PROGRAM pouPROFINETdiag
VAR
	iVal: WORD;
	tVal: WORD;
	tmask: WORD;
	state: UINT;
	i: UINT;
	decode:fb_decodeProfiNet;
	
	retvall: UDINT;
	idbGetConfSlaves: FB_EcGetConfSlaves;
	test: BOOL;
	testams: BOOL;
	a: UINT;
	tDiagScreenSize: UINT;
	tDiagScreenWidth: UINT;
	tDiagScreenPointer: UINT;
	testvalprofinet: PROFINETstate;
	
	detectFallingFault:F_TRIG;
END_VAR
VAR // added by the converter: edge detectors and wires of the graphical bodies
    _rt1, _rt2, _rt3, _rt4, _rt5 : R_TRIG;
END_VAR

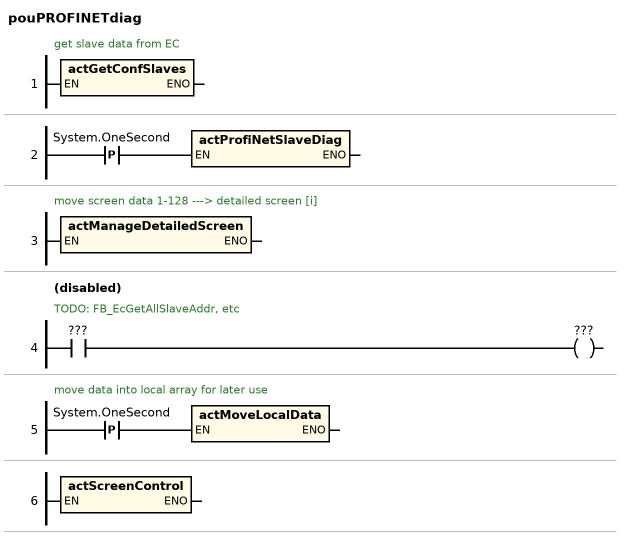
// NETWORK 1
// get slave data from EC
actGetConfSlaves();

// NETWORK 2
_rt1(CLK := System.OneSecond);
IF _rt1.Q THEN actProfiNetSlaveDiag(); END_IF

// NETWORK 3
// move screen data 1-128 ---> detailed screen [i]
actManageDetailedScreen();

// NETWORK 4 (disabled)
// TODO: FB_EcGetAllSlaveAddr, etc
// ??? := ???;

// NETWORK 5
// move data into local array for later use
_rt2(CLK := System.OneSecond);
IF _rt2.Q THEN actMoveLocalData(); END_IF

// NETWORK 6
actScreenControl();

ACTION actGetConfSlaves:
// NETWORK 1
// use System.OneSecond to slow down reading

// NETWORK 2
// get additional profinet info via ADS
END_ACTION

ACTION actManageDetailedScreen:
//get max value of diag number
ProfiNetDiag.detailDiagNum := MAX(ProfiNetDiag.detailDiagNum, 1);

IF System.PulseOneSecond THEN
	retvall := MEMCPY( destAddr	:=ADR(ProfiNetDiag.detailDiag),
						srcAddr :=ADR(ProfiNetDiag.diagScreen[ProfiNetDiag.detailDiagNum]),
						n		:=SIZEOF(ProfiNetDiag.detailDiag)
						);
END_IF
END_ACTION

ACTION actMoveLocalData:
//move data from FB_EcGetConfSlaves (etherCATdiag.arryEcConfSlaveInfo) to data for HMI

FOR a := 1 TO ProfiNetDiag.maxNumProfiNetSlaves DO
	//this is for detailed command for profinet, via ADS?
	//ProfiNetDiag.ProfiNetslaveDiag[a].ConfigData := ProfiNetDiag.arryEcConfSlaveInfo[a];

END_FOR
END_ACTION

ACTION actProfiNetSlaveDiag:



FOR i := 1 TO  ProfiNetDiag.maxNumProfiNetSlaves DO //

////////////////////////////////////////////////////////////////
//test write value
//TODO: REMOVE
ProfiNetDiag.RawProfiNetStateDiag[i] := testvalprofinet; 
ProfiNetDiag.ProfiNetslaveDiag[i].SlaveNumber := i;
//ProfiNetDiag.EtherCATslaveDiag[i].crcCount.portA := i;
/////////////////////////////////////////////////////////////////


//move temp data from scan to temp declarations
decode(iVal:=ProfiNetDiag.RawProfiNetStateDiag[i],iVal2:=16#0000); //confirm where iVal2 comes from (PN diag)
ProfiNetDiag.ProfiNetslaveDiag[i].currentState.state := decode.state;
ProfiNetDiag.ProfiNetslaveDiag[i].currentState.suffix := decode.suffix; //isnt really a suffix, just keeping the name the same


	//check values for fault
	//current state
	IF ProfiNetDiag.ProfiNetslaveDiag[i].currentState.state <> PROFINETstate.NoError THEN //EtherCATstate.OP 
		ProfiNetDiag.ProfiNetslaveDiag[i].currentState.isFault := TRUE;
		ELSE
		ProfiNetDiag.ProfiNetslaveDiag[i].currentState.isFault := FALSE;	
	END_IF
	

	//record outer box
	//record previous state, latching 
	detectFallingFault(CLK:=ProfiNetDiag.ProfiNetslaveDiag[i].currentState.isFault);
		IF detectFallingFault.Q THEN
		//at this time, record the current state in the historical state
		ProfiNetDiag.ProfiNetslaveDiag[i].historicalState.state := ProfiNetDiag.ProfiNetslaveDiag[i].currentState.state;
		ProfiNetDiag.ProfiNetslaveDiag[i].historicalState.suffix := ProfiNetDiag.ProfiNetslaveDiag[i].currentState.suffix;
		ProfiNetDiag.ProfiNetslaveDiag[i].historicalState.isFault := TRUE;
		ProfiNetDiag.ProfiNetslaveDiag[i].historicalState.colour := ProfiNetDiag.ProfiNetslaveDiag[i].currentState.colour;
	END_IF
	
	//clear inner box when fault is resolved
	IF 	ProfiNetDiag.ProfiNetslaveDiag[i].currentState.isFault = FALSE AND
	   gHMIButtons.btnReset THEN
	   ProfiNetDiag.ProfiNetslaveDiag[i].historicalState.isFault := FALSE;
	  	ProfiNetDiag.ProfiNetslaveDiag[i].historicalState.state := PROFINETstate.NoError;
		ProfiNetDiag.ProfiNetslaveDiag[i].historicalState.suffix := ProfiNetSuffix.NoDiagnostics;
	ProfiNetDiag.ProfiNetslaveDiag[i].historicalState.colour := HMIColour.colourGreen;

	END_IF
	

			//check if any suffix fault exits
			IF ProfiNetDiag.ProfiNetslaveDiag[i].currentState.state > 0 THEN
						
				//check suffix
				CASE ProfiNetDiag.ProfiNetslaveDiag[i].currentState.state OF 
				PROFINETstate.NoError								: 	ProfiNetDiag.ProfiNetslaveDiag[i].currentState.colour := HMIColour.colourGreen;
				PROFINETstate.StateInBoot							: 	ProfiNetDiag.ProfiNetslaveDiag[i].currentState.colour := HMIColour.colourRed;
				PROFINETstate.DeviceNotFound						: 	ProfiNetDiag.ProfiNetslaveDiag[i].currentState.colour := HMIColour.colourRed;
				PROFINETstate.StationNameNotUnique					: 	ProfiNetDiag.ProfiNetslaveDiag[i].currentState.colour := HMIColour.colourRed;
				PROFINETstate.IPCouldNotBeSet						: 	ProfiNetDiag.ProfiNetslaveDiag[i].currentState.colour := HMIColour.colourRed;
				PROFINETstate.IPConfict								: 	ProfiNetDiag.ProfiNetslaveDiag[i].currentState.colour := HMIColour.colourRed;
				PROFINETstate.DCPSetNotSuccessful					: 	ProfiNetDiag.ProfiNetslaveDiag[i].currentState.colour := HMIColour.colourRed;
				PROFINETstate.WatchdogError							: 	ProfiNetDiag.ProfiNetslaveDiag[i].currentState.colour := HMIColour.colourRed;
				PROFINETstate.DataholdError							: 	ProfiNetDiag.ProfiNetslaveDiag[i].currentState.colour := HMIColour.colourRed;
				PROFINETstate.RTC3SyncModeNotInit					: 	ProfiNetDiag.ProfiNetslaveDiag[i].currentState.colour := HMIColour.colourRed;
				PROFINETstate.ProfinetContLinkError					: 	ProfiNetDiag.ProfiNetslaveDiag[i].currentState.colour := HMIColour.colourRed;
				PROFINETstate.AliasnameNotUnique					: 	ProfiNetDiag.ProfiNetslaveDiag[i].currentState.colour := HMIColour.colourRed;
				PROFINETstate.AutoNameAssignNotPossibleWrongDevice	: 	ProfiNetDiag.ProfiNetslaveDiag[i].currentState.colour := HMIColour.colourRed;
				PROFINETstate.NoApplicationReady					: 	ProfiNetDiag.ProfiNetslaveDiag[i].currentState.colour := HMIColour.colourRed;
				PROFINETstate.ModuleDiffrence						: 	ProfiNetDiag.ProfiNetslaveDiag[i].currentState.colour := HMIColour.colourRed;
				PROFINETstate.InputCRInvalid						: 	ProfiNetDiag.ProfiNetslaveDiag[i].currentState.colour := HMIColour.colourRed;
				PROFINETstate.OutputCRInvalid						: 	ProfiNetDiag.ProfiNetslaveDiag[i].currentState.colour := HMIColour.colourRed;
				PROFINETstate.WCStateEtherCATframe_1				: 	ProfiNetDiag.ProfiNetslaveDiag[i].currentState.colour := HMIColour.colourRed;
				END_CASE;
				
			ELSE
				
				//otherwise check state to get green
				CASE ProfiNetDiag.ProfiNetslaveDiag[i].currentState.suffix OF 
				ProfiNetSuffix.NoDiagnostics							: 	ProfiNetDiag.ProfiNetslaveDiag[i].currentState.colour := HMIColour.colourGreen;
				ProfiNetSuffix.IOCAR_NotEstablished						: 	ProfiNetDiag.ProfiNetslaveDiag[i].currentState.colour := HMIColour.colourRed;
				ProfiNetSuffix.IOCAR_IsEstablished						: 	ProfiNetDiag.ProfiNetslaveDiag[i].currentState.colour := HMIColour.colourRed;
				ProfiNetSuffix.IOCAR_EstablishedNoApplicationReady		: 	ProfiNetDiag.ProfiNetslaveDiag[i].currentState.colour := HMIColour.colourRed;
				ProfiNetSuffix.IOCAR_EstablishedModuleDiffrence			: 	ProfiNetDiag.ProfiNetslaveDiag[i].currentState.colour := HMIColour.colourRed;
				ProfiNetSuffix.AlarmCR_DiagnosticAlarm					: 	ProfiNetDiag.ProfiNetslaveDiag[i].currentState.colour := HMIColour.colourRed;
				ProfiNetSuffix.InputCR_Invalid							: 	ProfiNetDiag.ProfiNetslaveDiag[i].currentState.colour := HMIColour.colourRed;
				ProfiNetSuffix.InputCR_ProviderInStop					: 	ProfiNetDiag.ProfiNetslaveDiag[i].currentState.colour := HMIColour.colourRed;
				ProfiNetSuffix.InputCR_ProblemIndicatorIsSet			: 	ProfiNetDiag.ProfiNetslaveDiag[i].currentState.colour := HMIColour.colourRed;
				ProfiNetSuffix.OutputCR_Invalid							: 	ProfiNetDiag.ProfiNetslaveDiag[i].currentState.colour := HMIColour.colourRed;
				ProfiNetSuffix.OutputCR_ProviderInStop					: 	ProfiNetDiag.ProfiNetslaveDiag[i].currentState.colour := HMIColour.colourRed;
				ProfiNetSuffix.OutputCR_ProblemIndicatorIsSet			: 	ProfiNetDiag.ProfiNetslaveDiag[i].currentState.colour := HMIColour.colourRed;
				END_CASE;
				
			END_IF
	
	
END_FOR
END_ACTION

ACTION actScreenControl:
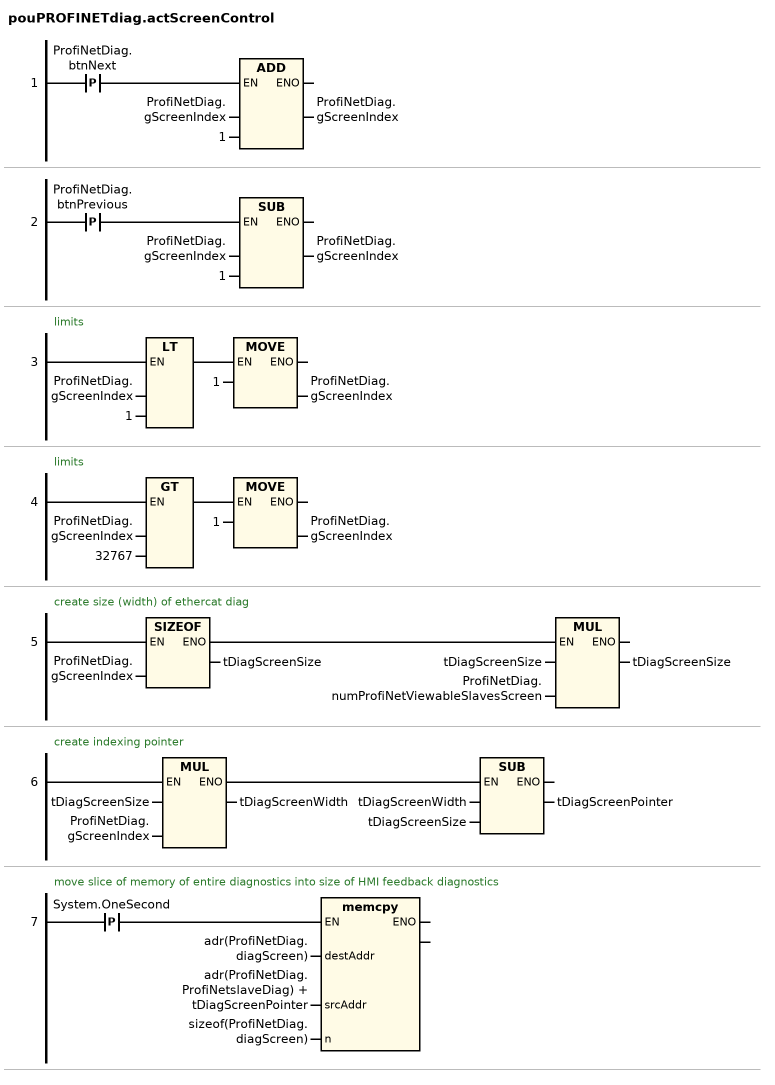
// NETWORK 1
_rt3(CLK := ProfiNetDiag.btnNext);
IF _rt3.Q THEN ProfiNetDiag.gScreenIndex := ProfiNetDiag.gScreenIndex + 1; END_IF

// NETWORK 2
_rt4(CLK := ProfiNetDiag.btnPrevious);
IF _rt4.Q THEN ProfiNetDiag.gScreenIndex := ProfiNetDiag.gScreenIndex - 1; END_IF

// NETWORK 3
// limits
IF ProfiNetDiag.gScreenIndex < 1 THEN ProfiNetDiag.gScreenIndex := 1; END_IF

// NETWORK 4
// limits
IF ProfiNetDiag.gScreenIndex > 32767 THEN ProfiNetDiag.gScreenIndex := 1; END_IF

// NETWORK 5
// create size (width) of ethercat diag
tDiagScreenSize := SIZEOF(ProfiNetDiag.gScreenIndex);
tDiagScreenSize := tDiagScreenSize * ProfiNetDiag.numProfiNetViewableSlavesScreen;

// NETWORK 6
// create indexing pointer
tDiagScreenWidth := tDiagScreenSize * ProfiNetDiag.gScreenIndex;
tDiagScreenPointer := tDiagScreenWidth - tDiagScreenSize;

// NETWORK 7
// move slice of memory of entire diagnostics into size of HMI feedback diagnostics
_rt5(CLK := System.OneSecond);
IF _rt5.Q THEN
    memcpy(destAddr := adr(ProfiNetDiag.diagScreen), srcAddr := adr(ProfiNetDiag.ProfiNetslaveDiag) + tDiagScreenPointer, n := sizeof(ProfiNetDiag.diagScreen));
END_IF
END_ACTION

END_PROGRAM

(* stored: Version 1.1.0.1, ProductVersion 3.1.4024.12
   POU pouPROFINETdiag: Id {6862f099-ed7c-4452-83ce-c9352fab3c19}, SpecialFunc None
   Action actGetConfSlaves: Id {12e9d60b-88c4-4151-a422-f7b5b76e7b29}
   Action actManageDetailedScreen: Id {69887705-3148-414b-900b-182318fc05ea}
   Action actMoveLocalData: Id {2663b4ef-3424-4ac8-9915-9b365465a05d}
   Action actProfiNetSlaveDiag: Id {b8897ab3-3f54-4d4c-9ca2-a475f035a090}
   Action actScreenControl: Id {21c06192-c051-48c4-ba33-4769c9e63527} *)
